// TIA Portal V20 export
// export: Created 2025-12-01T14:57:04.5162166Z, ExportSetting None, DisplayName Totally Integrated Automation Portal, DisplayVersion V20 Update 3, DisplayName TIA Portal Openness, DisplayVersion V20 Update 3, DisplayName TIA Portal Version Control Interface, DisplayVersion V20 Update 3, DisplayName STEP 7 Professional, DisplayVersion V20 Update 3, DisplayName STEP 7 Safety, DisplayVersion V20 Update 2, DisplayName WinCC Basic/Comfort/Advanced, DisplayVersion V20 Update 3, DisplayName WinCC Professional, DisplayVersion V20 Update 3, DisplayName WinCC Unified, DisplayVersion V20 Update 3
FUNCTION "FC791_GestorLlave" : Void   // FC791, LAD
{ S7_Optimized_Access := 'FALSE' }
AUTHOR : TRACKING
NAME : 20160411
VERSION : 3.1
// stored: AutoNumber false, SetENOAutomatically false
   VAR_INPUT
      NumLlave : UInt;
      Estado : Bool;
      MesaDeJDT02 : Bool;
   END_VAR
   VAR_OUTPUT
      Llave : "UDT_DatosLlave";
   END_VAR
   VAR_TEMP
      PunteroEventos : DWord;
      DBEventos : Word;
      NumDBEventos : UInt;
      MaxBytesDeEventos : UInt;
      NumBytes : UInt;
      Offset : UInt;   // Offset donde esta el Primer Dispositivo
      ValorTMP : UDInt;
      ValorReturn : Int;
   END_VAR
BEGIN

NETWORK
TITLE = Inicializar
////////////////////////////////////////////////////////////////////////////
// --- Inicializar Variables


////////////////////////////////////////////////////////////////////////////
// --- Control Numero de Dispositivo

      L     #NumLlave;
      L     1;
      <I;
      JC    FinalFuncion;  // Ha superado el minimo
      L     #NumLlave;
      L     "CTE_MaxDispositivosLlave";
      >I;
      JC    FinalFuncion;  // Ha superado el maximo



NETWORK
TITLE = Acciones
////////////////////////////////////////////////////////////////////////////
// --- Cambio de estado de la llave ?

      SET;
      A     #Estado;
      AN    "DB839_DispositivosVarios".DispoLlave[#NumLlave].EstadoActual;
      JC    CambioDeEstado_Llave;

      SET;
      AN    #Estado;
      A     "DB839_DispositivosVarios".DispoLlave[#NumLlave].EstadoActual;
      JC    CambioDeEstado_Llave;


////////////////////////////////////////////////////////////////////////////
// --- Mirar si hay peticion de Estado de Llave

      SET;
      A     "DB839_DispositivosVarios".DispoLlave[#NumLlave].RefrescoDatos;
      JC    EnviarEvento_RefrescoDeDatos;  // Hay Peticion de Esatdo ?
      JU    FinalFuncion;  // No Hay Peticion de estado



////////////////////////////////////////////////////////////////////////////
// --- Ha cambiado de estado la Llave

CambioDeEstado_Llave:NOP   0;
      SET;
      A     #Estado;  // Guardar el estado de la Llave
      =     "DB839_DispositivosVarios".DispoLlave[#NumLlave].EstadoActual;

      SET;
      S     "DB839_DispositivosVarios".DispoLlave[#NumLlave].RefrescoDatos;  // Activar la Peticion de Estado de la Llave

      JU    EnviarEvento_RefrescoDeDatos;  // Mandar nuevo evento de Estado de Llave



NETWORK
TITLE = Evento de Estado de la Llave
EnviarEvento_RefrescoDeDatos:NOP   0;

////////////////////////////////////////////////////////////////////////////
// ---   Formateo del Evento de Estado del Dispositivo
// ---   * Mirar si hay sitio para generar el nuevo evento
// ---       * Inicializo NumBytes y Puntero al DB de Eventos Generados
// ---       * Calcula el tamaño de bytes que hay en el DB de Eventos Generados
// ---       * Comprobar si hay sitio para un evento más
// ---   * Formatear el evento de Estado de las Llaves
////////////////////////////////////////////////////////////////////////////



////////////////////////////////////////////////////////////////////////////
// --- Inicio --> Pertenece a JDT 02 (Por defecto Pertenece a JDT01)

      L     "JDT1_NDB_EventosEmi";
      T     #DBEventos;
      T     #NumDBEventos;
      L     "JDT1_MaxBytes";
      T     #MaxBytesDeEventos;

      SET;
      AN    #MesaDeJDT02;
      JC    NoPerteneceJDT02;

      L     "JDT2_NDB_EventosEmi";
      T     #DBEventos;
      T     #NumDBEventos;
      L     "JDT2_MaxBytes";
      T     #MaxBytesDeEventos;

NoPerteneceJDT02:NOP   0;
// --- Fin --> Pertenece a JDT 02
////////////////////////////////////////////////////////////////////////////



////////////////////////////////////////////////////////////////////////////
// --- Mirar si hay sitio para generar un evento más

      L     0;
      T     #NumBytes;  // Inicializo el numero de Bytes
      T     #PunteroEventos;  // Inicializo el puntero de Eventos Generados

Inicio_BusquedaFinalEventos:NOP   0;
      OPN   DB [#DBEventos];  // Calcula el tamaño de bytes que hay en el DB
      L     DBB [#PunteroEventos];
      L     0;
      ==I;
      JC    Fin_BusquedaFinalEventos;  // Buscamos el final del DB = 0

      OPN   DB [#DBEventos];
      L     DBB [#PunteroEventos];
      L     ' ';
      ==I;
      JC    Fin_BusquedaFinalEventos;  // Buscamos el final del DB = ' '

      L     #PunteroEventos;  // Incremento de P#1.0
      L     P#1.0;
      +D;
      T     #PunteroEventos;

      JU    Inicio_BusquedaFinalEventos;  // Continuar con el siguiente posicion

Fin_BusquedaFinalEventos:NOP   0;
      L     #PunteroEventos;  // Sacamos el NumBytes Escritos
      SRD   3;
      T     #NumBytes;

      L     #NumBytes;  // Miramos si hay sitio
      L     #MaxBytesDeEventos;  // Max. que se pueden emitir, parametro
      >I;
      JC    FinalFuncion;  // No se pueden generar más eventos


////////////////////////////////////////////////////////////////////////////
// --- Formatear el evento de Estado del Dispositivo

      L     #PunteroEventos;
      LAR2;  // Puntero al DB de Eventos Generados

      TAR2;  // Mirar si es el primer evento de la lista
      L     0;
      ==I;
      JC    NoEsInicio_ListaDeEventos;  // Es el primero

      OPN   DB [#DBEventos];
      L     ',';  // Separador entre eventos ','
      T     DBB [AR2, P#0.0];
      +AR2  P#1.0;

NoEsInicio_ListaDeEventos:NOP   0;
      OPN   DB [#DBEventos];  // DB de Eventos Generados (A Emitir)
      L     '{';  // Inicio de Evento '{'
      T     DBB [AR2, P#0.0];
      +AR2  P#1.0;


////////////////////////////////////////////////////////////////////////////
      L     'STAT';  // --- Evento 'STAT'
      T     DBD [AR2, P#0.0];
      +AR2  P#4.0;


////////////////////////////////////////////////////////////////////////////
      OPN   DB [#DBEventos];
      L     '[';
      T     DBB [AR2, P#0.0];
      L     'TIPO';
      T     DBD [AR2, P#1.0];
      L     ']';
      T     DBB [AR2, P#5.0];
      +AR2  P#6.0;

      OPN   DB [#DBEventos];
      L     'LLAV';  // Tipo Llave
      T     DBD [AR2, P#0.0];
      +AR2  P#4.0;


////////////////////////////////////////////////////////////////////////////
      L     '[';
      T     DBB [AR2, P#0.0];
      L     'NUME';
      T     DBD [AR2, P#1.0];
      L     ']';
      T     DBB [AR2, P#5.0];
      +AR2  P#6.0;

      L     "CTE_OffsetMesa";
      L     #NumLlave;  // Numero de la Llave
      +I;
      T     #ValorTMP;

// --- Convertir Valor a ASCII - Numero de la Baliza
      TAR2;
      SRD   3;
      T     #NumBytes;  // Miro que offset tiene la String

      CALL  "FC893_Obtener_StringDelAtributo"
      ( DB_String := #NumDBEventos,
        OffsetIni := #NumBytes,
        Valor     := #ValorTMP,
        OffsetFin := #Offset
      );  // Llamo a ObtenerStrinAtributo

      L     #Offset;
      SLD   3;
      LAR2;  // Recupero que offset tiene la String

// --- Ya esta convertido el Valor a ASCII

////////////////////////////////////////////////////////////////////////////
      OPN   DB [#DBEventos];
      L     '[';
      T     DBB [AR2, P#0.0];
      L     'ACTI';
      T     DBD [AR2, P#1.0];
      L     ']';
      T     DBB [AR2, P#5.0];
      +AR2  P#6.0;

      L     'SI';
      SET;
      A     "DB839_DispositivosVarios".DispoLlave[#NumLlave].EstadoActual;  // Activo Llave ?
      JC    EstaActiva_Llave;
      L     'NO';
EstaActiva_Llave:NOP   0;
      OPN   DB [#DBEventos];
      T     DBW [AR2, P#0.0];
      +AR2  P#2.0;


////////////////////////////////////////////////////////////////////////////
      OPN   DB [#DBEventos];
      L     '[';
      T     DBB [AR2, P#0.0];
      L     'HABI';
      T     DBD [AR2, P#1.0];
      L     ']';
      T     DBB [AR2, P#5.0];
      +AR2  P#6.0;

      L     'SI';
      SET;
      A     "DB839_DispositivosVarios".DispoLlave[#NumLlave].Habilitado;  // Habilitado ?
      JC    EstaDesHabilitada_Llave;
      L     'NO';
EstaDesHabilitada_Llave:NOP   0;
      OPN   DB [#DBEventos];
      T     DBW [AR2, P#0.0];
      +AR2  P#2.0;


////////////////////////////////////////////////////////////////////////////
      OPN   DB [#DBEventos];  // DB de Eventos Generados (A Emitir)
      L     '}';  // --- Fin de Evento '}'
      T     DBB [AR2, P#0.0];
      +AR2  P#1.0;



////////////////////////////////////////////////////////////////////////////
// --- Final del Evento

      SET;
      R     "DB839_DispositivosVarios".DispoLlave[#NumLlave].RefrescoDatos;  // Activar la Peticion de Estado de la Baliza

      JU    FinalFuncion;  //Final del Formateo del Elento



NETWORK
TITLE = Final de la Función
////////////////////////////////////////////////////////////////////////////
FinalFuncion:NOP   0;

      CALL  BLKMOV
      ( SRCBLK  := "DB839_DispositivosVarios".DispoLlave[#NumLlave],
        RET_VAL := #ValorReturn,
        DSTBLK  := #Llave
      );


END_FUNCTION
